(* PLC project CoDeSys External Library Template, WAGO e!COCKPIT e!COCKPIT, author 3S - Smart Software Solutions GmbH *)
(* stored: creationDateTime 2019-10-29T12:22:40.8732585, version 3.5.5.30, modificationDateTime 2019-10-24T14:40:07.960949, organization 3S - Smart Software Solutions GmbH *)
(* Library project template with all possible element types, docu and a sample project structure *)

FUNCTION fnKomunikatDaneZnajdzPorownajZapisz : BOOL
  VAR_INPUT
    sKomunikat : alSTRINGKomunikat;  (* Ramka z IZE *)
    sAtrybut : STRING;  (* Atrybut do wyszukania w ramce *)
  END_VAR
  VAR_IN_OUT
    rAtrybutWartosc : REAL;  (* Wartość atrybutu w sterowniku *)
    sDane : STRING;  (* Dane do wysłania w ramce *)
  END_VAR
  VAR_OUTPUT
    xAtrybutZapisz : BOOL;  (* Trigger zapisu wartości atrybutu do urządzenia *)
  END_VAR
  VAR
    sAtrybutWartoscRamka : STRING;  (* Wartość atrybutu z ramki *)
    rAtrybutWartoscRamka : REAL;  (* Wartość atrybutu z ramki *)
  END_VAR

            (*			
Autor:					Artur Wyszomirski, 2019-06-04 
Prawa majątkowe: 		Solwena Sp. z o.o., 
Aktualizacje:			
Opis:					Porównanie wartości atrybutu z ramki przychodzącej z IZE z wartością atrybutu zapisaną w sterowniku (urządzeniu). Jeśli wartość jest różna, triggerowana jest zmienna xAtrybutZapisz (zapis wartości do urządzenia).
						W przeciwnym wypadku nazwa atrybutu i jego wartość przpisywane są do sDane (czyli pola danych ramki A, którą sterownik wyśle w odpowiedzi do IZE) 
*)

sAtrybutWartoscRamka := fnKomunikatDaneSzukajWartosci(sKomunikat, sAtrybut);
// Jeśli wartość atrybutu została odnaleziona w ramce.
IF sAtrybutWartoscRamka <> '' THEN
	rAtrybutWartoscRamka := (STRING_TO_REAL(sAtrybutWartoscRamka));
	// Jeśli wartość różni się od dotychczasowej, zapisz ją. W przeciwnym wypadku doklej wartość do ramki A.
	IF rAtrybutWartoscRamka <> rAtrybutWartosc THEN
		rAtrybutWartosc := rAtrybutWartoscRamka;
		xAtrybutZapisz := TRUE;
	ELSE
		IF sDane <> '' THEN
			sDane := CONCAT(sDane , ';');
		END_IF					
		sDane := CONCAT(sDane , sAtrybut);
		sDane := CONCAT(sDane , sAtrybutWartoscRamka);
	END_IF
END_IF

          
END_FUNCTION
